(* CoDeSys 2.3 library: CMP_OC_W10.lib *)
(* Libraries: STANDARD.LIB 5.6.98 11:03:02 *)

(* POU MAIN, LD *)
PROGRAM MAIN
VAR
END_VAR
_LD_ (* Ladder Diagram *)
_END_LD_
END_PROGRAM

(* POU CMP_OC_W1, FBD *)
FUNCTIONBLOCK CMP_OC_W1

VAR_INPUT
	WORD_1: WORD;		(*WORD 1*)
	END_VAR


VAR_OUTPUT
	BZ_OUTPUT_BOOL : BOOL;
END_VAR


VAR
	OUT_1: BOOL;
END_VAR
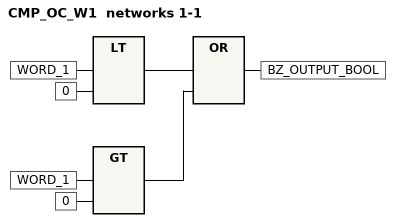
_FBD_ (* Function Block Diagram *)
NETWORK 1
	OR(LT(WORD_1, 0), GT(WORD_1, 0)) => BZ_OUTPUT_BOOL
_END_FBD_
(* the same logic as Structured Text *)
(* Network 1 *)
BZ_OUTPUT_BOOL := (WORD_1 < 0) OR (WORD_1 > 0);
END_FUNCTION_BLOCK

(* POU CMP_OC_W10, FBD *)
FUNCTIONBLOCK CMP_OC_W10

VAR_INPUT
	WORD_1: WORD;		(*WORD 1*)
	WORD_2: WORD;		(*WORD 2*)
	WORD_3: WORD;		(*WORD 3*)
	WORD_4: WORD;		(*WORD 4*)
	WORD_5: WORD;		(*WORD 5*)
	WORD_6: WORD;		(*WORD 6*)
	WORD_7: WORD;		(*WORD 7*)
	WORD_8: WORD;		(*WORD 8*)
	WORD_9: WORD;		(*WORD 9*)
	WORD_10: WORD;	(*WORD 10*)
END_VAR


VAR_OUTPUT
	BZ_OUTPUT_BOOL : BOOL;
END_VAR


VAR
	OUT_1: BOOL;
	OUT_2: BOOL;
	OUT_3: BOOL;
	OUT_4: BOOL;
	OUT_5: BOOL;
	OUT_6: BOOL;
	OUT_7: BOOL;
	OUT_8: BOOL;
	OUT_9: BOOL;
	OUT_10: BOOL;

END_VAR
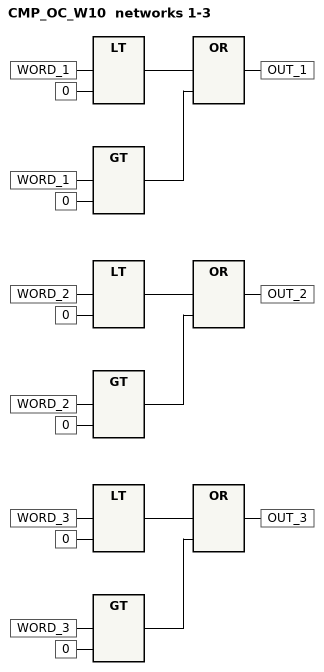
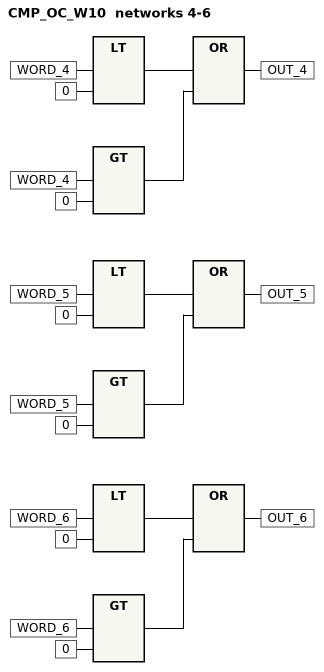
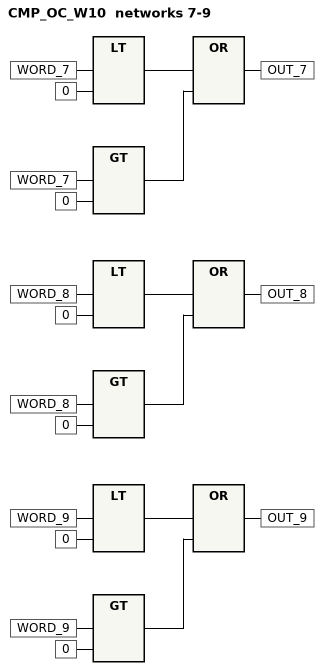
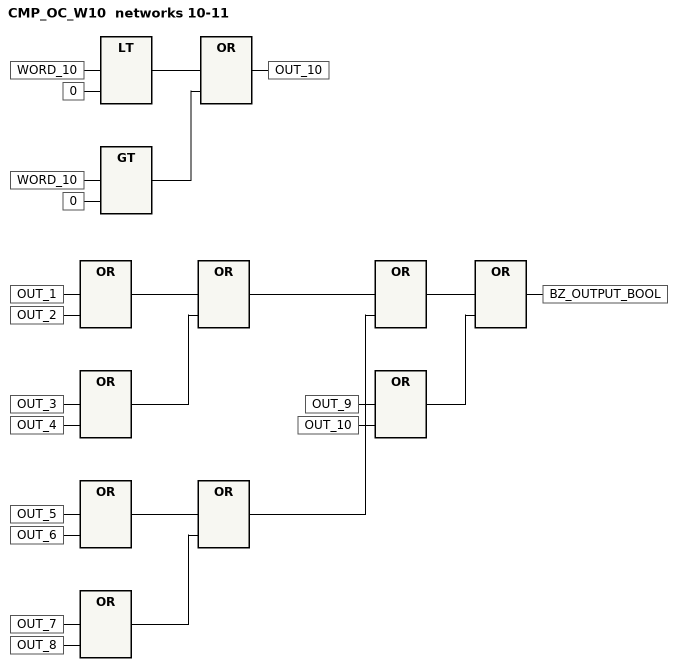
_FBD_ (* Function Block Diagram *)
NETWORK 1
	OR(LT(WORD_1, 0), GT(WORD_1, 0)) => OUT_1
NETWORK 2
	OR(LT(WORD_2, 0), GT(WORD_2, 0)) => OUT_2
NETWORK 3
	OR(LT(WORD_3, 0), GT(WORD_3, 0)) => OUT_3
NETWORK 4
	OR(LT(WORD_4, 0), GT(WORD_4, 0)) => OUT_4
NETWORK 5
	OR(LT(WORD_5, 0), GT(WORD_5, 0)) => OUT_5
NETWORK 6
	OR(LT(WORD_6, 0), GT(WORD_6, 0)) => OUT_6
NETWORK 7
	OR(LT(WORD_7, 0), GT(WORD_7, 0)) => OUT_7
NETWORK 8
	OR(LT(WORD_8, 0), GT(WORD_8, 0)) => OUT_8
NETWORK 9
	OR(LT(WORD_9, 0), GT(WORD_9, 0)) => OUT_9
NETWORK 10
	OR(LT(WORD_10, 0), GT(WORD_10, 0)) => OUT_10
NETWORK 11
	OR(OR(OR(OR(OUT_1, OUT_2), OR(OUT_3, OUT_4)), OR(OR(OUT_5, OUT_6), OR(OUT_7, OUT_8))), OR(OUT_9, OUT_10)) => BZ_OUTPUT_BOOL
_END_FBD_
(* the same logic as Structured Text *)
(* Network 1 *)
OUT_1 := (WORD_1 < 0) OR (WORD_1 > 0);
(* Network 2 *)
OUT_2 := (WORD_2 < 0) OR (WORD_2 > 0);
(* Network 3 *)
OUT_3 := (WORD_3 < 0) OR (WORD_3 > 0);
(* Network 4 *)
OUT_4 := (WORD_4 < 0) OR (WORD_4 > 0);
(* Network 5 *)
OUT_5 := (WORD_5 < 0) OR (WORD_5 > 0);
(* Network 6 *)
OUT_6 := (WORD_6 < 0) OR (WORD_6 > 0);
(* Network 7 *)
OUT_7 := (WORD_7 < 0) OR (WORD_7 > 0);
(* Network 8 *)
OUT_8 := (WORD_8 < 0) OR (WORD_8 > 0);
(* Network 9 *)
OUT_9 := (WORD_9 < 0) OR (WORD_9 > 0);
(* Network 10 *)
OUT_10 := (WORD_10 < 0) OR (WORD_10 > 0);
(* Network 11 *)
BZ_OUTPUT_BOOL := (((OUT_1 OR OUT_2) OR (OUT_3 OR OUT_4)) OR ((OUT_5 OR OUT_6) OR (OUT_7 OR OUT_8))) OR (OUT_9 OR OUT_10);
END_FUNCTION_BLOCK

(* POU CMP_OC_W2, FBD *)
FUNCTIONBLOCK CMP_OC_W2

VAR_INPUT
	WORD_1: WORD;		(*WORD 1*)
	WORD_2: WORD;		(*WORD 2*)
	END_VAR


VAR_OUTPUT
	BZ_OUTPUT_BOOL : BOOL;
END_VAR


VAR
	OUT_1: BOOL;
	OUT_2: BOOL;
END_VAR
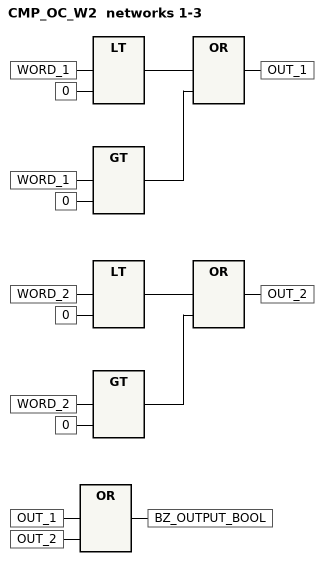
_FBD_ (* Function Block Diagram *)
NETWORK 1
	OR(LT(WORD_1, 0), GT(WORD_1, 0)) => OUT_1
NETWORK 2
	OR(LT(WORD_2, 0), GT(WORD_2, 0)) => OUT_2
NETWORK 3
	OR(OUT_1, OUT_2) => BZ_OUTPUT_BOOL
_END_FBD_
(* the same logic as Structured Text *)
(* Network 1 *)
OUT_1 := (WORD_1 < 0) OR (WORD_1 > 0);
(* Network 2 *)
OUT_2 := (WORD_2 < 0) OR (WORD_2 > 0);
(* Network 3 *)
BZ_OUTPUT_BOOL := OUT_1 OR OUT_2;
END_FUNCTION_BLOCK

(* POU CMP_OC_W3, FBD *)
FUNCTIONBLOCK CMP_OC_W3

VAR_INPUT
	WORD_1: WORD;		(*WORD 1*)
	WORD_2: WORD;		(*WORD 2*)
	WORD_3: WORD;		(*WORD 3*)
	END_VAR


VAR_OUTPUT
	BZ_OUTPUT_BOOL : BOOL;
END_VAR


VAR
	OUT_1: BOOL;
	OUT_2: BOOL;
	OUT_3: BOOL;
END_VAR
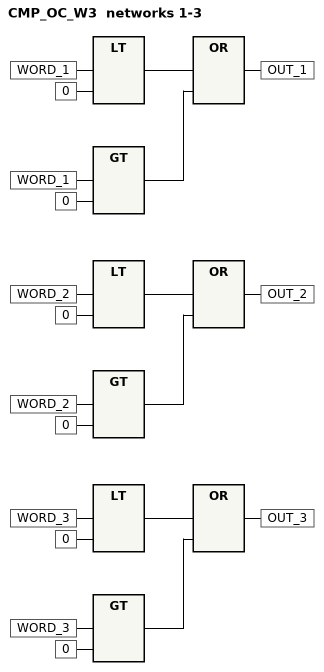
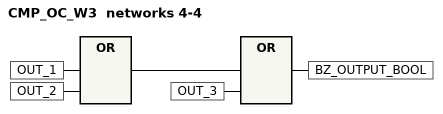
_FBD_ (* Function Block Diagram *)
NETWORK 1
	OR(LT(WORD_1, 0), GT(WORD_1, 0)) => OUT_1
NETWORK 2
	OR(LT(WORD_2, 0), GT(WORD_2, 0)) => OUT_2
NETWORK 3
	OR(LT(WORD_3, 0), GT(WORD_3, 0)) => OUT_3
NETWORK 4
	OR(OR(OUT_1, OUT_2), OUT_3) => BZ_OUTPUT_BOOL
_END_FBD_
(* the same logic as Structured Text *)
(* Network 1 *)
OUT_1 := (WORD_1 < 0) OR (WORD_1 > 0);
(* Network 2 *)
OUT_2 := (WORD_2 < 0) OR (WORD_2 > 0);
(* Network 3 *)
OUT_3 := (WORD_3 < 0) OR (WORD_3 > 0);
(* Network 4 *)
BZ_OUTPUT_BOOL := (OUT_1 OR OUT_2) OR OUT_3;
END_FUNCTION_BLOCK

(* POU CMP_OC_W4, FBD *)
FUNCTIONBLOCK CMP_OC_W4

VAR_INPUT
	WORD_1: WORD;		(*WORD 1*)
	WORD_2: WORD;		(*WORD 2*)
	WORD_3: WORD;		(*WORD 3*)
	WORD_4: WORD;		(*WORD 4*)
	END_VAR


VAR_OUTPUT
	BZ_OUTPUT_BOOL : BOOL;
END_VAR


VAR
	OUT_1: BOOL;
	OUT_2: BOOL;
	OUT_3: BOOL;
	OUT_4: BOOL;
END_VAR
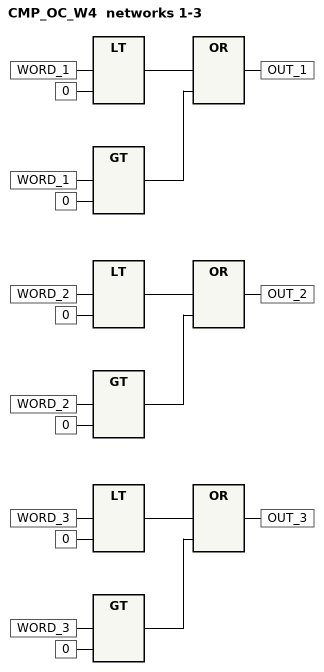
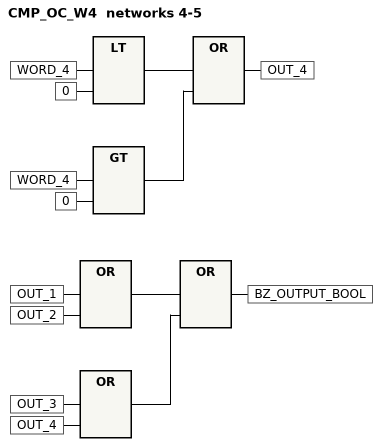
_FBD_ (* Function Block Diagram *)
NETWORK 1
	OR(LT(WORD_1, 0), GT(WORD_1, 0)) => OUT_1
NETWORK 2
	OR(LT(WORD_2, 0), GT(WORD_2, 0)) => OUT_2
NETWORK 3
	OR(LT(WORD_3, 0), GT(WORD_3, 0)) => OUT_3
NETWORK 4
	OR(LT(WORD_4, 0), GT(WORD_4, 0)) => OUT_4
NETWORK 5
	OR(OR(OUT_1, OUT_2), OR(OUT_3, OUT_4)) => BZ_OUTPUT_BOOL
_END_FBD_
(* the same logic as Structured Text *)
(* Network 1 *)
OUT_1 := (WORD_1 < 0) OR (WORD_1 > 0);
(* Network 2 *)
OUT_2 := (WORD_2 < 0) OR (WORD_2 > 0);
(* Network 3 *)
OUT_3 := (WORD_3 < 0) OR (WORD_3 > 0);
(* Network 4 *)
OUT_4 := (WORD_4 < 0) OR (WORD_4 > 0);
(* Network 5 *)
BZ_OUTPUT_BOOL := (OUT_1 OR OUT_2) OR (OUT_3 OR OUT_4);
END_FUNCTION_BLOCK

(* POU CMP_OC_W5, FBD *)
FUNCTIONBLOCK CMP_OC_W5

VAR_INPUT
	WORD_1: WORD;		(*WORD 1*)
	WORD_2: WORD;		(*WORD 2*)
	WORD_3: WORD;		(*WORD 3*)
	WORD_4: WORD;		(*WORD 4*)
	WORD_5: WORD;		(*WORD 5*)
END_VAR


VAR_OUTPUT
	BZ_OUTPUT_BOOL : BOOL;
END_VAR


VAR
	OUT_1: BOOL;
	OUT_2: BOOL;
	OUT_3: BOOL;
	OUT_4: BOOL;
	OUT_5: BOOL;
END_VAR
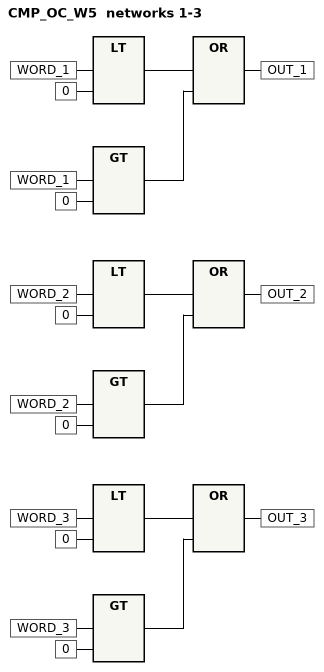
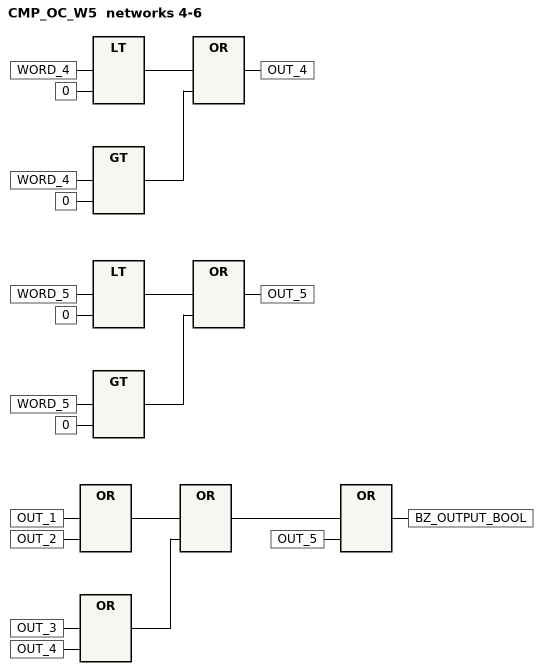
_FBD_ (* Function Block Diagram *)
NETWORK 1
	OR(LT(WORD_1, 0), GT(WORD_1, 0)) => OUT_1
NETWORK 2
	OR(LT(WORD_2, 0), GT(WORD_2, 0)) => OUT_2
NETWORK 3
	OR(LT(WORD_3, 0), GT(WORD_3, 0)) => OUT_3
NETWORK 4
	OR(LT(WORD_4, 0), GT(WORD_4, 0)) => OUT_4
NETWORK 5
	OR(LT(WORD_5, 0), GT(WORD_5, 0)) => OUT_5
NETWORK 6
	OR(OR(OR(OUT_1, OUT_2), OR(OUT_3, OUT_4)), OUT_5) => BZ_OUTPUT_BOOL
_END_FBD_
(* the same logic as Structured Text *)
(* Network 1 *)
OUT_1 := (WORD_1 < 0) OR (WORD_1 > 0);
(* Network 2 *)
OUT_2 := (WORD_2 < 0) OR (WORD_2 > 0);
(* Network 3 *)
OUT_3 := (WORD_3 < 0) OR (WORD_3 > 0);
(* Network 4 *)
OUT_4 := (WORD_4 < 0) OR (WORD_4 > 0);
(* Network 5 *)
OUT_5 := (WORD_5 < 0) OR (WORD_5 > 0);
(* Network 6 *)
BZ_OUTPUT_BOOL := ((OUT_1 OR OUT_2) OR (OUT_3 OR OUT_4)) OR OUT_5;
END_FUNCTION_BLOCK

(* POU CMP_OC_W6, FBD *)
FUNCTIONBLOCK CMP_OC_W6

VAR_INPUT
	WORD_1: WORD;		(*WORD 1*)
	WORD_2: WORD;		(*WORD 2*)
	WORD_3: WORD;		(*WORD 3*)
	WORD_4: WORD;		(*WORD 4*)
	WORD_5: WORD;		(*WORD 5*)
	WORD_6: WORD;		(*WORD 6*)
END_VAR


VAR_OUTPUT
	BZ_OUTPUT_BOOL : BOOL;
END_VAR


VAR
	OUT_1: BOOL;
	OUT_2: BOOL;
	OUT_3: BOOL;
	OUT_4: BOOL;
	OUT_5: BOOL;
	OUT_6: BOOL;
END_VAR
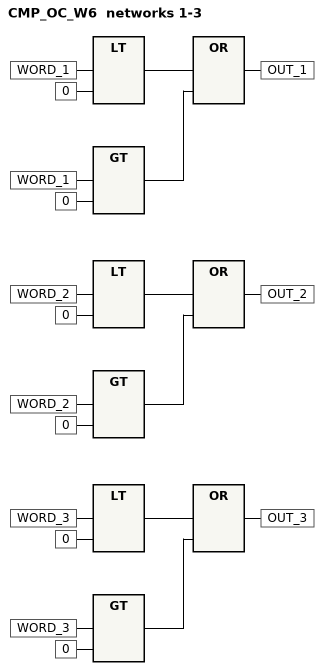
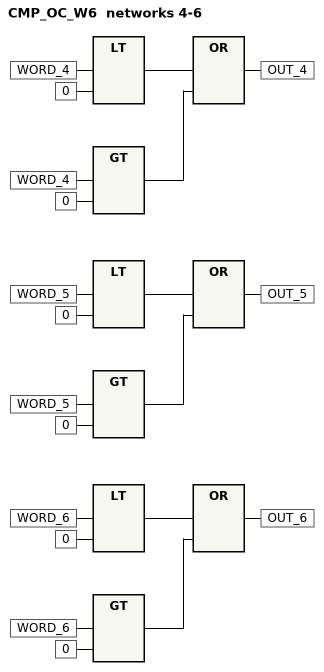
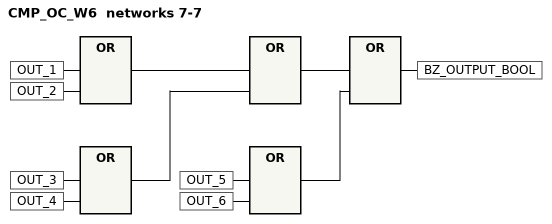
_FBD_ (* Function Block Diagram *)
NETWORK 1
	OR(LT(WORD_1, 0), GT(WORD_1, 0)) => OUT_1
NETWORK 2
	OR(LT(WORD_2, 0), GT(WORD_2, 0)) => OUT_2
NETWORK 3
	OR(LT(WORD_3, 0), GT(WORD_3, 0)) => OUT_3
NETWORK 4
	OR(LT(WORD_4, 0), GT(WORD_4, 0)) => OUT_4
NETWORK 5
	OR(LT(WORD_5, 0), GT(WORD_5, 0)) => OUT_5
NETWORK 6
	OR(LT(WORD_6, 0), GT(WORD_6, 0)) => OUT_6
NETWORK 7
	OR(OR(OR(OUT_1, OUT_2), OR(OUT_3, OUT_4)), OR(OUT_5, OUT_6)) => BZ_OUTPUT_BOOL
_END_FBD_
(* the same logic as Structured Text *)
(* Network 1 *)
OUT_1 := (WORD_1 < 0) OR (WORD_1 > 0);
(* Network 2 *)
OUT_2 := (WORD_2 < 0) OR (WORD_2 > 0);
(* Network 3 *)
OUT_3 := (WORD_3 < 0) OR (WORD_3 > 0);
(* Network 4 *)
OUT_4 := (WORD_4 < 0) OR (WORD_4 > 0);
(* Network 5 *)
OUT_5 := (WORD_5 < 0) OR (WORD_5 > 0);
(* Network 6 *)
OUT_6 := (WORD_6 < 0) OR (WORD_6 > 0);
(* Network 7 *)
BZ_OUTPUT_BOOL := ((OUT_1 OR OUT_2) OR (OUT_3 OR OUT_4)) OR (OUT_5 OR OUT_6);
END_FUNCTION_BLOCK

(* POU CMP_OC_W7, FBD *)
FUNCTIONBLOCK CMP_OC_W7

VAR_INPUT
	WORD_1: WORD;		(*WORD 1*)
	WORD_2: WORD;		(*WORD 2*)
	WORD_3: WORD;		(*WORD 3*)
	WORD_4: WORD;		(*WORD 4*)
	WORD_5: WORD;		(*WORD 5*)
	WORD_6: WORD;		(*WORD 6*)
	WORD_7: WORD;		(*WORD 7*)
END_VAR


VAR_OUTPUT
	BZ_OUTPUT_BOOL : BOOL;
END_VAR


VAR
	OUT_1: BOOL;
	OUT_2: BOOL;
	OUT_3: BOOL;
	OUT_4: BOOL;
	OUT_5: BOOL;
	OUT_6: BOOL;
	OUT_7: BOOL;
END_VAR
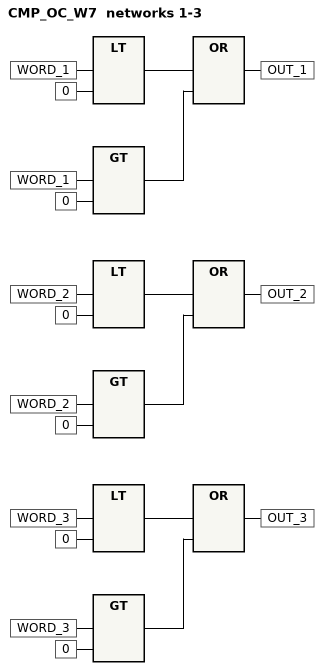
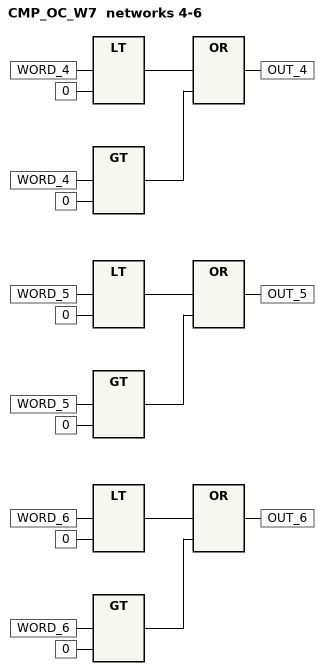
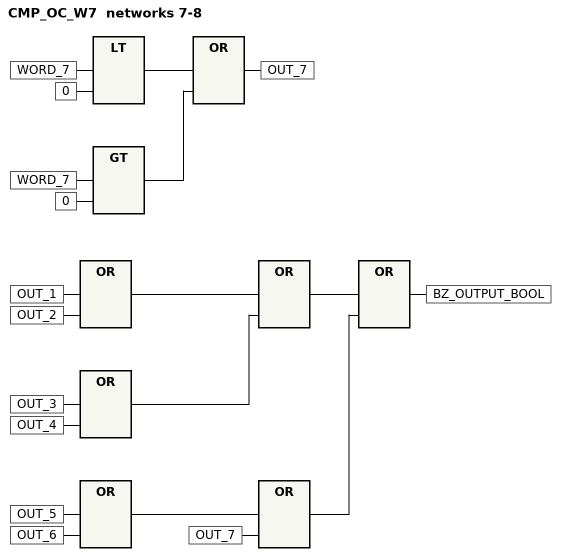
_FBD_ (* Function Block Diagram *)
NETWORK 1
	OR(LT(WORD_1, 0), GT(WORD_1, 0)) => OUT_1
NETWORK 2
	OR(LT(WORD_2, 0), GT(WORD_2, 0)) => OUT_2
NETWORK 3
	OR(LT(WORD_3, 0), GT(WORD_3, 0)) => OUT_3
NETWORK 4
	OR(LT(WORD_4, 0), GT(WORD_4, 0)) => OUT_4
NETWORK 5
	OR(LT(WORD_5, 0), GT(WORD_5, 0)) => OUT_5
NETWORK 6
	OR(LT(WORD_6, 0), GT(WORD_6, 0)) => OUT_6
NETWORK 7
	OR(LT(WORD_7, 0), GT(WORD_7, 0)) => OUT_7
NETWORK 8
	OR(OR(OR(OUT_1, OUT_2), OR(OUT_3, OUT_4)), OR(OR(OUT_5, OUT_6), OUT_7)) => BZ_OUTPUT_BOOL
_END_FBD_
(* the same logic as Structured Text *)
(* Network 1 *)
OUT_1 := (WORD_1 < 0) OR (WORD_1 > 0);
(* Network 2 *)
OUT_2 := (WORD_2 < 0) OR (WORD_2 > 0);
(* Network 3 *)
OUT_3 := (WORD_3 < 0) OR (WORD_3 > 0);
(* Network 4 *)
OUT_4 := (WORD_4 < 0) OR (WORD_4 > 0);
(* Network 5 *)
OUT_5 := (WORD_5 < 0) OR (WORD_5 > 0);
(* Network 6 *)
OUT_6 := (WORD_6 < 0) OR (WORD_6 > 0);
(* Network 7 *)
OUT_7 := (WORD_7 < 0) OR (WORD_7 > 0);
(* Network 8 *)
BZ_OUTPUT_BOOL := ((OUT_1 OR OUT_2) OR (OUT_3 OR OUT_4)) OR ((OUT_5 OR OUT_6) OR OUT_7);
END_FUNCTION_BLOCK

(* POU CMP_OC_W8, FBD *)
FUNCTIONBLOCK CMP_OC_W8

VAR_INPUT
	WORD_1: WORD;		(*WORD 1*)
	WORD_2: WORD;		(*WORD 2*)
	WORD_3: WORD;		(*WORD 3*)
	WORD_4: WORD;		(*WORD 4*)
	WORD_5: WORD;		(*WORD 5*)
	WORD_6: WORD;		(*WORD 6*)
	WORD_7: WORD;		(*WORD 7*)
	WORD_8: WORD;		(*WORD 8*)
END_VAR


VAR_OUTPUT
	BZ_OUTPUT_BOOL : BOOL;
END_VAR


VAR
	OUT_1: BOOL;
	OUT_2: BOOL;
	OUT_3: BOOL;
	OUT_4: BOOL;
	OUT_5: BOOL;
	OUT_6: BOOL;
	OUT_7: BOOL;
	OUT_8: BOOL;
END_VAR
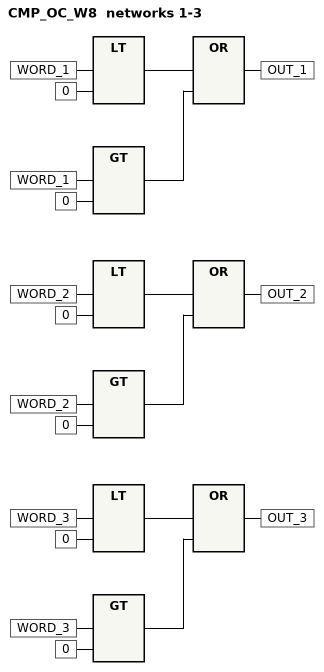
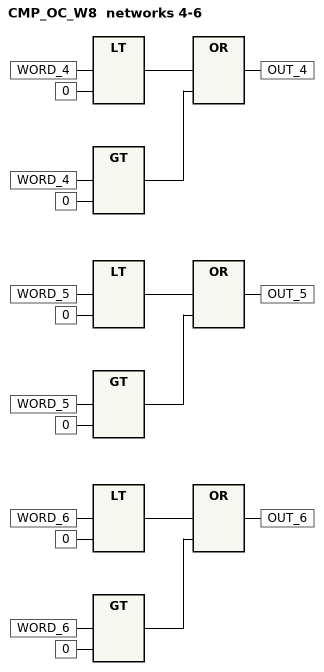
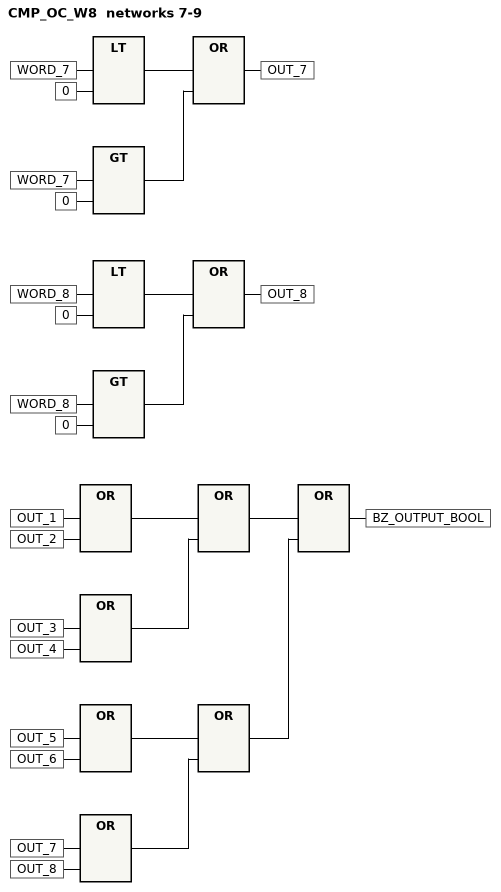
_FBD_ (* Function Block Diagram *)
NETWORK 1
	OR(LT(WORD_1, 0), GT(WORD_1, 0)) => OUT_1
NETWORK 2
	OR(LT(WORD_2, 0), GT(WORD_2, 0)) => OUT_2
NETWORK 3
	OR(LT(WORD_3, 0), GT(WORD_3, 0)) => OUT_3
NETWORK 4
	OR(LT(WORD_4, 0), GT(WORD_4, 0)) => OUT_4
NETWORK 5
	OR(LT(WORD_5, 0), GT(WORD_5, 0)) => OUT_5
NETWORK 6
	OR(LT(WORD_6, 0), GT(WORD_6, 0)) => OUT_6
NETWORK 7
	OR(LT(WORD_7, 0), GT(WORD_7, 0)) => OUT_7
NETWORK 8
	OR(LT(WORD_8, 0), GT(WORD_8, 0)) => OUT_8
NETWORK 9
	OR(OR(OR(OUT_1, OUT_2), OR(OUT_3, OUT_4)), OR(OR(OUT_5, OUT_6), OR(OUT_7, OUT_8))) => BZ_OUTPUT_BOOL
_END_FBD_
(* the same logic as Structured Text *)
(* Network 1 *)
OUT_1 := (WORD_1 < 0) OR (WORD_1 > 0);
(* Network 2 *)
OUT_2 := (WORD_2 < 0) OR (WORD_2 > 0);
(* Network 3 *)
OUT_3 := (WORD_3 < 0) OR (WORD_3 > 0);
(* Network 4 *)
OUT_4 := (WORD_4 < 0) OR (WORD_4 > 0);
(* Network 5 *)
OUT_5 := (WORD_5 < 0) OR (WORD_5 > 0);
(* Network 6 *)
OUT_6 := (WORD_6 < 0) OR (WORD_6 > 0);
(* Network 7 *)
OUT_7 := (WORD_7 < 0) OR (WORD_7 > 0);
(* Network 8 *)
OUT_8 := (WORD_8 < 0) OR (WORD_8 > 0);
(* Network 9 *)
BZ_OUTPUT_BOOL := ((OUT_1 OR OUT_2) OR (OUT_3 OR OUT_4)) OR ((OUT_5 OR OUT_6) OR (OUT_7 OR OUT_8));
END_FUNCTION_BLOCK

(* POU CMP_OC_W9, FBD *)
FUNCTIONBLOCK CMP_OC_W9

VAR_INPUT
	WORD_1: WORD;		(*WORD 1*)
	WORD_2: WORD;		(*WORD 2*)
	WORD_3: WORD;		(*WORD 3*)
	WORD_4: WORD;		(*WORD 4*)
	WORD_5: WORD;		(*WORD 5*)
	WORD_6: WORD;		(*WORD 6*)
	WORD_7: WORD;		(*WORD 7*)
	WORD_8: WORD;		(*WORD 8*)
	WORD_9: WORD;		(*WORD 9*)
END_VAR


VAR_OUTPUT
	BZ_OUTPUT_BOOL : BOOL;
END_VAR


VAR
	OUT_1: BOOL;
	OUT_2: BOOL;
	OUT_3: BOOL;
	OUT_4: BOOL;
	OUT_5: BOOL;
	OUT_6: BOOL;
	OUT_7: BOOL;
	OUT_8: BOOL;
	OUT_9: BOOL;
END_VAR
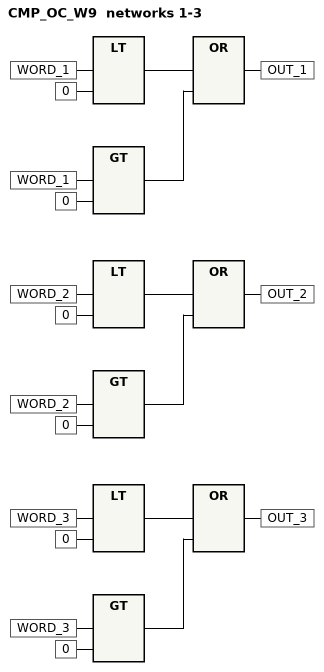
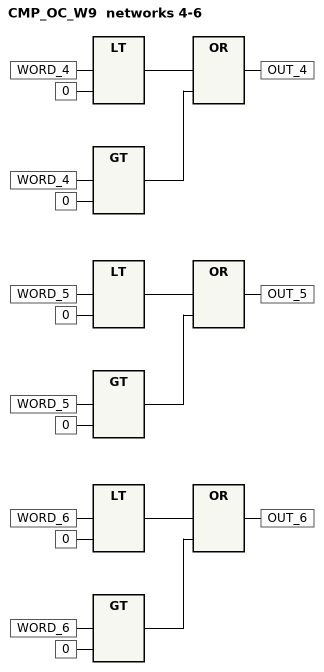
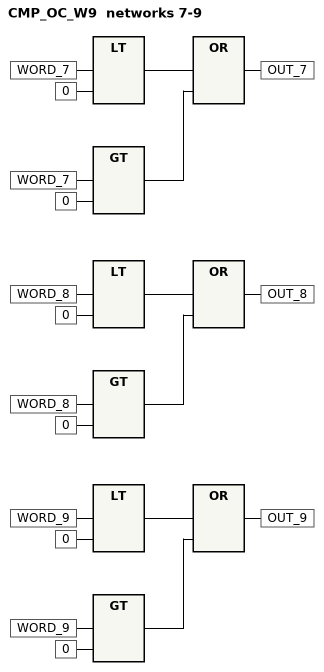
